FUNCTION_BLOCK FB_Home_Sequence
VAR_INPUT
END_VAR
VAR_OUTPUT
	HomeDone : BOOL;
END_VAR
VAR
	
nHome : INT := 0;
	FbLagHomie: MC_StepBlockLagBasedDetection;
	FB_MOVE_BRO: MC_MoveAbsolute;
END_VAR

CASE nHome OF


0:
	HomeDone := FALSE;

		FbLagHomie(
				Axis:= , //y axis
				Parameter:= MC_HomingParameter , 
				Execute:= TRUE, 
				Direction:= MC_Home_Direction.mcPositiveDirection, 
				Velocity:= , //SPEEEED
				Acceleration:= , 
				Deceleration:= , 
				Jerk:= , 
				DetectionVelocityLimit:= , //low SPEEED
				DetectionVelocityTime:= , //T#1 
				TimeLimit:= , // 5 seconds please
				DistanceLimit:= ,//  idk 10k bro 
				TorqueLimit:= , // torque limit safe 
				LagLimit:= , // what ever is just a bit higher then the lag when the motor starts 
				BufferMode:= , 
				Options:= , 
				Done:=  ,
				Busy=> , 
				Active=> , 
				CommandAborted=> , 
				Error=> , 
				ErrorID=> , 
				RecordedPosition=> );
	
 1: 

      	FB_MOVE_BRO(
				Axis:= , //Y-axis
				Execute:=TRUE, 
				Position:= 100, // plus or minus figure it out bro 
				Velocity:= , //Low and Slow
				Acceleration:= , 
				Deceleration:= , 
				Jerk:= , 
				BufferMode:= , 
				Options:= , 
				Done=> ,
				Busy=> , 
				Active=> , 
				CommandAborted=> , 
				Error=> , 
				ErrorID=> );
		IF FB_MOVE_BRO.Done THEN
			HomeDone := TRUE;
		END_IF

END_FUNCTION_BLOCK

(* stored: Version 1.1.0.1, ProductVersion 3.1.4024.11
   POU FB_Home_Sequence: Id {0ccc3fcd-e1a1-4e4f-b16c-6c129ce5ceec}, SpecialFunc None *)
